// SIMATIC S7-200 project (STEP 7-Micro/WIN), CPU 221 REL 01.10

ORGANIZATION_BLOCK MAIN:OB1
TITLE=PROGRAM COMMENTS
BEGIN
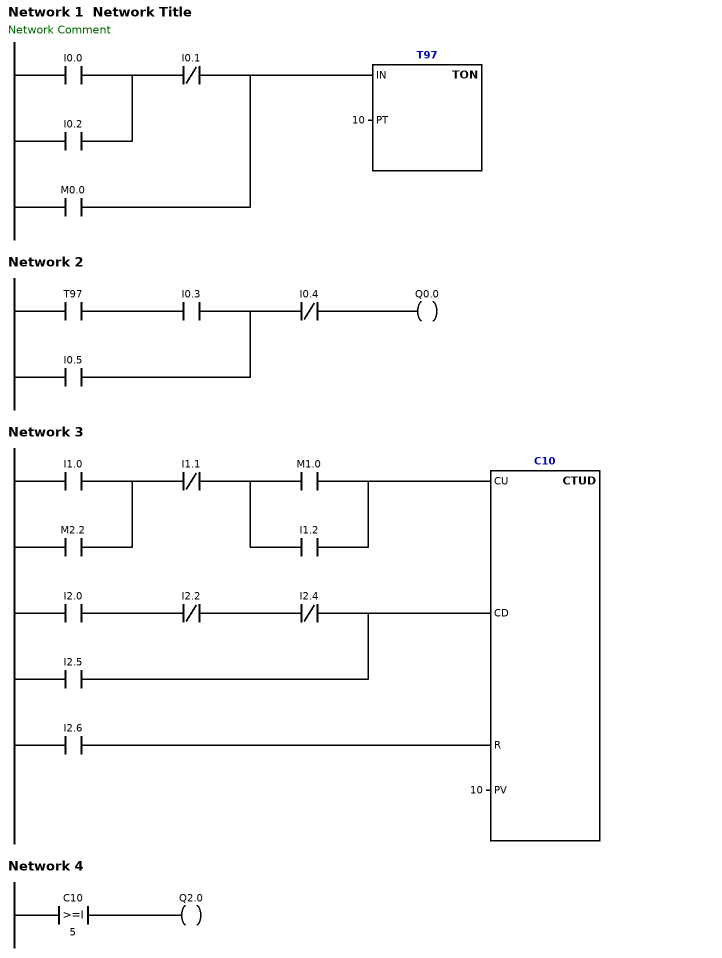
Network 1 // Network Title
// Network Comment
LD     I0.0
O      I0.2
AN     I0.1
O      M0.0
TON    T97, 10
Network 2
LD     T97
A      I0.3
O      I0.5
AN     I0.4
=      Q0.0
Network 3
LD     I1.0
O      M2.2
AN     I1.1
LD     M1.0
O      I1.2
ALD
LD     I2.0
AN     I2.2
AN     I2.4
O      I2.5
LD     I2.6
CTUD   C10, 10
Network 4
LDW>=  C10, 5
=      Q2.0
END_ORGANIZATION_BLOCK
